PROGRAM main
VAR
	Start AT %IX0.0 : bool;
	Stop AT %IX0.1 : bool;
	SystemActive AT %QX0.0 : bool;
END_VAR

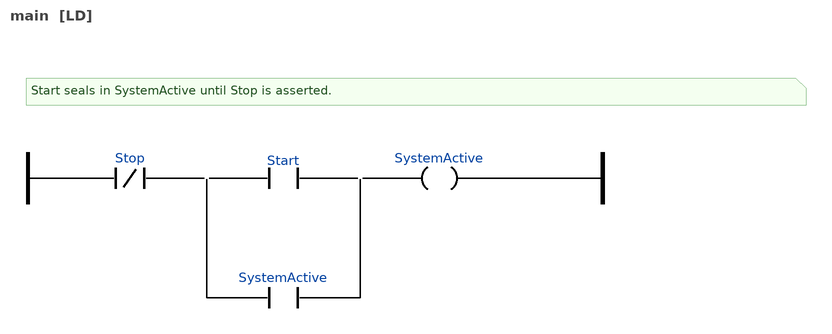
(* LD diagram, written out as Structured Text *)
(* Start seals in SystemActive until Stop is asserted. *)
SystemActive := NOT Stop AND (Start OR SystemActive);
END_PROGRAM
